PROGRAM TESTS
VAR
  DateTime_TEST : DateTime_TEST;
  HelperFunctions_TEST : ConvertAnyToString_TEST;
  DynamicStringBuffer_TEST : DynamicStringBuffer_TEST;
  TestWrapper : TestWrapper_NET();
END_VAR

TcUnit.RUN();

TestWrapper();

END_PROGRAM

(* stored: Version 1.1.0.1, ProductVersion 3.1.4026.8
   POU TESTS: Id {379526ca-9719-4af5-b69e-537f4c5508c9}, SpecialFunc None *)
